Staubli VAL3: Product.dtx

bool bExit
bool bListRefresh
bool bUserRefresh
mdesc mNomSpeed
num nPage
num nSelected
public string sDeli[2]
  [0] = "A"
  [1] = "C"
public string sFileList
string sFolder = "Disk://Traj/"
string sItem = "paodpe"
string sList[2]
  [0] = "paodpe"
  [1] = "popo"
string sOutputFolder = "Disk://Traj/"
string sPathList
num nPrdIndex
string sNewPath
string sProductList
string sPrd
